ABB RAPID module: CalibData.modx

MODULE CalibData
    PERS tooldata TCP_KruvikeerajaABB_V2:=[TRUE,[[-337.5,-0.733,119.997],[0.707107,0,-0.707107,0]],[1,[0,0,1],[1,0,0,0],0,0,0]];
ENDMODULE
